FUNCTION F_SYSTEM_BoolToBArcodeType : E_CodeType
VAR_INPUT
	bPackBarcode		: BOOL;
	bInterimBarcode	: BOOL;
	bOuterBarcode		: BOOL;
	bCaseBarcode		: BOOL;
END_VAR
VAR
END_VAR

IF bPackBarcode THEN
	F_SYSTEM_BoolToBArcodeType := E_PACK;
ELSIF bInterimBarcode THEN
	F_SYSTEM_BoolToBArcodeType := E_INTERIM;
ELSIF bOuterBarcode THEN
	F_SYSTEM_BoolToBArcodeType := E_OUTER;
ELSIF bCaseBarcode THEN
	F_SYSTEM_BoolToBArcodeType := E_CASE;
ELSE
	F_SYSTEM_BoolToBArcodeType := E_NONE;
END_IF

END_FUNCTION

(* stored: Version 1.1.0.1, ProductVersion 3.1.4024.15
   POU F_SYSTEM_BoolToBArcodeType: Id {76ca1352-19b8-4418-b20c-72383926ae55}, SpecialFunc None *)
